//==================================================================================================
//							Beckhoff Automation Poland
//									23.05.2018
//	Blok funkcyjny kontroli luzownika w silniku podpietym do AX5000. Przewaga ForceLock
//	Datatype:		ENUM (INT16)
//	Enum Value:		0 (0x00): 	Release_force
//					1 (0x01): 	Force_lock
//					2 (0x02): 	Force_unlock
//
// 	v1.1	|| TC v 3.1.4022.16	|| - optymalizacja kodu
//  v1.0	|| TC v 3.1.4022.16	|| - pierwsza wersja
//==================================================================================================
FUNCTION_BLOCK FB_HoldingBrakeCtrlAX5000
VAR_INPUT
	bForceLock 						: BOOL;								// 
	bForceUnlock					: BOOL;								// 
END_VAR
VAR_OUTPUT
	bBusy							: BOOL;
	bError							: BOOL; 							// General error: parameter or CoE read.
																		// If bError = TRUE and bInitialized = FALSE - error during read motor data.
																		// If bError = TRUE and bInitialized = TRUE and (iAdsErrId <> 0 or iCANopenErrId <> 0) then I2T read error
																		// If bError = TRUE and bInitialized = TRUE and iAdsErrId = 0 and iCANopenErrId = 0 then parameter error: rTorqueLimit outside permitted range rTorqueLimitLow..rTorqueLimitHigh or Empty stDriveRef
	iAdsErrId						: UINT;								// Forwarded output FB_SoEWrite
	iSecErrId						: UINT;								// Forwarded output FB_SoEWrite
END_VAR
VAR_IN_OUT
	Axis							: AXIS_REF;
END_VAR
VAR
	bExecute						: BOOL;
	iMotorBrakeForce				: INT;								// 0 - Release_force, 1 - Force_lock, 2 - Force_unlock
	fbSoEWrite						: FB_SoEWrite;
	rtForceLock						: R_TRIG;
	rtForceUnlock					: R_TRIG;
	ftForceLock						: F_TRIG;
	ftForceUnlock					: F_TRIG;
END_VAR

{region "Call triggers"}
//======================= Call triggers =========================
rtForceLock(CLK:= bForceLock);
ftForceLock(CLK:= bForceLock);
rtForceUnlock(CLK:= bForceUnlock);
ftForceUnlock(CLK:= bForceUnlock);
bExecute								:= rtForceLock.Q OR ftForceLock.Q OR rtForceUnlock.Q OR ftForceUnlock.Q;
//===============================================================
{endregion}
{region "Main code"}
//========================= Main code ===========================
IF bExecute THEN
	iMotorBrakeForce 						:= 0;										// Clear value
	iMotorBrakeForce.1 						:= bForceUnlock;							// Set force unlock bit
	iMotorBrakeForce 						:= SEL(bForceLock, iMotorBrakeForce, 1);	// Set force lock bit, it has higher priority than unlock
END_IF
	 
fbSoEWrite(
	NetId			:= '' , 
	Idn				:= P_0_IDN + 96 , 
	Element			:= 16#40 , 
	pSrcBuf			:= ADR(iMotorBrakeForce), 
	BufLen			:= SIZEOF(iMotorBrakeForce) , 
	Execute			:= bExecute , 
	Timeout			:= T#2S, 
	Axis			:= Axis , 
	Busy			=> bBusy , 
	Error			=> bError, 
	AdsErrId		=> iAdsErrId, 
	SercosErrId		=> iSecErrId );
//===============================================================
{endregion}

END_FUNCTION_BLOCK

(* stored: Version 1.1.0.1, ProductVersion 3.1.4026.13, FileIdentifier 2b54be542da9aeb12c4fb40fab00f34829536606, FileSignature 34e1c7af544d29c23fef9e3877958b6e2c4f6be76dc41c51d00a3d365f91165c96ce8a36b248068e37ed13284f1f7dc84553d275439e9050f236110f15a2dca41f57bcccc6667f7bf7a5d39a6df015a2c9b72f4d02df7e717b902258e3bf901259cdc8a00b564d8032f5612f0b05cb8db6215792be0597d0493e02f2448ec03810118a39ad9b202f37a9c9330672381731406d94b6d45dc51b7a6c6c67d7650f4455b363d8beeb730807f465411c5080c2693e196c05ebe74fd5dbdb9144ad7e0eb43d88a8ce7cce5edd91a879fadd19cc9c01157c62f3f294bf3a83c2f1e848971033ec248256373abef4d521cecb6bd172ea670ebe5cd908175287f6704cdc
   POU FB_HoldingBrakeCtrlAX5000: Id {c1953c0a-f8e1-44b4-8946-27e90a6eeff4}, SpecialFunc None *)
